{attribute addProperty BoxType "EL3068-0000-0019"}
{attribute addProperty Id "AI_Standard_ChannelAT %I*ARRAY[0..7] OF AI_Standard_Channel_F16A160D256320WcStateAT %I*WcState_98A4DF7520.250InfoDataAT %I*InfoData_BC63D37F80100"}
{attribute addProperty CRC "2754435194"}
{attribute addProperty SizeInBites "338"}
{attribute addProperty SizeInBytes "42.25"}
TYPE EL3068_EA60A077 :
STRUCT
	{attribute addProperty Name "AI_Standard_Channel"}
	AI_Standard_Channel : ARRAY[0..7] OF AI_Standard_Channel_F16A160D;
	{attribute addProperty Name "WcState"}
	WcState : WcState_98A4DF75;
	{attribute addProperty Name "InfoData"}
	InfoData : InfoData_BC63D37F;
END_STRUCT
END_TYPE

(* stored: Version 1.2.0.0, ProductVersion 3.1.4024.9
   DUT EL3068_EA60A077: Id {29c2bf5f-f888-441d-91ca-474bc27b859b} *)
